Fanuc KAREL source: kt00112.KL

-- PROVISIONAL review KL for V1013-1; original PC SHA256 ee5d539785db829db32efe9c112e133a1ba4283cbaa3f53c75ee38083c2e6d3b
-- Incomplete behavior may be omitted. Consult companion uncertainty JSON. Do not deploy.
PROGRAM KT00112
%NOLOCKGROUP
VAR
  R1 : REAL
  OUT : REAL
-- UNRESOLVED_DECL H2 type=002017
BEGIN
  -- UNRESOLVED_PC offsets 5-16; opcodes 2E,23
  -- UNRESOLVED_PC offsets 21-35; opcodes 2E,22,9D,33,B4
  -- UNRESOLVED_PC offsets 40-63; opcodes 21,22,9D,33,B3,64,6C,23
  -- UNRESOLVED_PC offsets 68-72; opcodes 7F
END KT00112
